FUNCTION_BLOCK QualityFailFilter (* Tolerancia de tempo para a falha de canal por qualidade do sinal (por instancia do AnalogInput) *)
  (* Standard: 61499-2 *)
  (* Version 1.0, 10/7/2026, Claude/Hidryco, Schneider Electric, Rev0 - Falha de canal (qualidade ruim/incerta) so e confirmada se persistir por FailDelay; 0 = imediato (comportamento anterior). Usado no AnalogInput (40FT05). *)
  PACKAGE SE.Nereda;
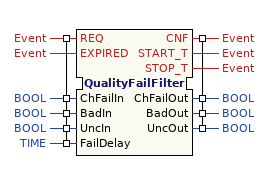
  EVENT_INPUT
    REQ WITH ChFailIn, BadIn, UncIn, FailDelay; (* Nova avaliacao da falha de canal *)
    EXPIRED; (* Fim do tempo de tolerancia (E_DELAY.EO) *)
  END_EVENT
  EVENT_OUTPUT
    CNF WITH ChFailOut, BadOut, UncOut; (* Falha de canal filtrada (a cada avaliacao) *)
    START_T; (* Inicia o temporizador de tolerancia (E_DELAY.START) *)
    STOP_T; (* Para o temporizador de tolerancia (E_DELAY.STOP) *)
  END_EVENT
  VAR_INPUT
    ChFailIn : BOOL; (* Falha de canal bruta (OR de qualidade ruim, qualidade incerta e falha do AnalogInputBase) *)
    BadIn : BOOL; (* Qualidade ruim (aiSignalDecode.Bad) *)
    UncIn : BOOL; (* Qualidade incerta (aiSignalDecode.Uncertain) *)
    FailDelay : TIME; (* Tolerancia: a falha so e confirmada se durar este tempo (0 = imediato) *)
  END_VAR
  VAR_OUTPUT
    ChFailOut : BOOL; (* Falha de canal confirmada *)
    BadOut : BOOL; (* Qualidade ruim com a falha confirmada (alarme BadQuality) *)
    UncOut : BOOL; (* Qualidade incerta com a falha confirmada (alarme UncertainQuality) *)
  END_VAR
  VAR
    Timing : BOOL; (* Temporizador de tolerancia contando *)
    Confirmed : BOOL; (* Falha confirmada *)
    FromTimer : BOOL; (* Avaliacao disparada pelo fim do tempo *)
    DoStart : BOOL;
    DoStop : BOOL;
  END_VAR
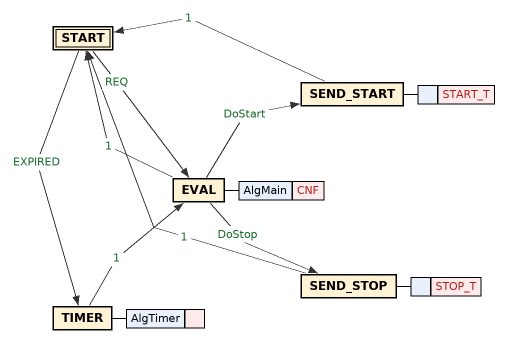
  EC_STATES
    START; (* Initial State *)
    EVAL : AlgMain -> CNF; (* Avalia e publica *)
    TIMER : AlgTimer; (* Fim do tempo de tolerancia *)
    SEND_START : -> START_T;
    SEND_STOP : -> STOP_T;
  END_STATES
  EC_TRANSITIONS
    START TO EVAL := REQ;
    START TO TIMER := EXPIRED;
    TIMER TO EVAL := 1;
    EVAL TO SEND_START := DoStart;
    EVAL TO SEND_STOP := DoStop;
    EVAL TO START := 1;
    SEND_START TO START := 1;
    SEND_STOP TO START := 1;
  END_TRANSITIONS
  ALGORITHM AlgMain IN ST: (* Tolerancia da falha de canal *)
;
(* QualityFailFilter - tolerancia para a falha de canal (qualidade do sinal)
   ChFailIn = OR bruto (qualidade ruim, qualidade incerta, falha do AnalogInputBase).
   A falha so e confirmada se ficar presente sem interrupcao durante FailDelay.
   FailDelay = 0 (padrao): confirma na hora - mesmo comportamento de antes.
   Ao normalizar (ChFailIn = FALSE), limpa na hora e para o temporizador.
   BadOut / UncOut = qualidade ruim / incerta, so com a falha confirmada (alarmes da lista). *)
DoStart := FALSE;
DoStop := FALSE;
IF NOT ChFailIn THEN
    IF Timing THEN
        DoStop := TRUE;
    END_IF;
    Timing := FALSE;
    Confirmed := FALSE;
ELSIF NOT Confirmed THEN
    IF FailDelay <= T#0s THEN
        IF Timing THEN
            DoStop := TRUE;
        END_IF;
        Timing := FALSE;
        Confirmed := TRUE;
    ELSIF FromTimer AND Timing THEN
        Timing := FALSE;
        Confirmed := TRUE;
    ELSIF NOT Timing THEN
        Timing := TRUE;
        DoStart := TRUE;
    END_IF;
END_IF;
FromTimer := FALSE;
ChFailOut := Confirmed;
BadOut := BadIn AND Confirmed;
UncOut := UncIn AND Confirmed;
  END_ALGORITHM
  ALGORITHM AlgTimer IN ST: (* Fim do tempo de tolerancia *)
;
(* fim do tempo de tolerancia (E_DELAY.EO) *)
FromTimer := TRUE;
  END_ALGORITHM
END_FUNCTION_BLOCK
